RoboDK station: bp.rdk

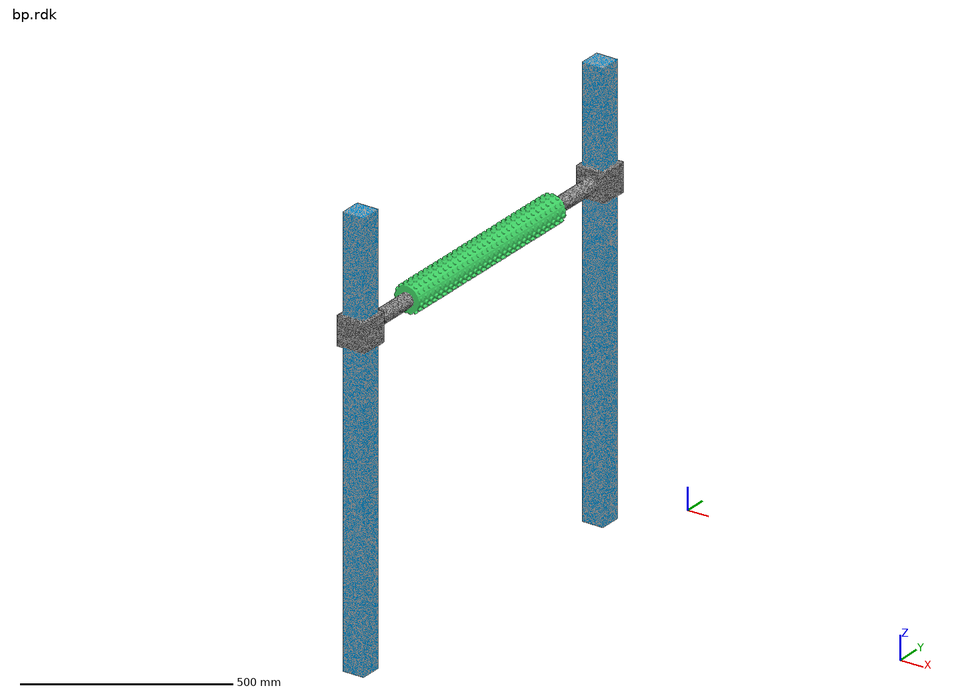
[picture v0: the station drawn from its stored meshes, robots at their saved joint values, targets as dots, program paths as lines]
Station bp (saved by RoboDK 5.8.0). Poses are relative to the parent item; angles as X-Y-Z fixed-axis rotations.
  - frame Mi Mecanismo Base at (0, 1000, 0) mm
    - robot Mi Mecanismo: 2 axes
        modified DH rows (alpha deg, a mm, theta deg, d mm): -90, 0, 0, 1000 linear; 90, 0, 0, 0
        base shift (-140, 0, 40) mm, rotated rx 90 ry 0 rz 0 deg
        joint limits [-200, 0] to [110, 360]; home [0, 0]; saved at [-148.96, 186.52]
